{attribute 'linkalways'} 
{attribute 'no_explicit_call' := 'This FB is a CLASS and must be accessed using methods or properties'}
{attribute 'enable_dynamic_creation'}
FUNCTION_BLOCK Node_F_VN_EnclosingTriangle EXTENDS VisionNode
VAR
    ipPointSet : _ITcVnContainer;
    aTriangleVertices : _TcVnArray3_Point2_REAL;
    fArea : _LREAL(0.0);
    hrPrev : _HRESULT(S_OK);
	hresult : _HRESULT(S_OK);
END_VAR

METHOD PUBLIC  Clone : I_Node
VAR
	pNode : POINTER TO Node_F_VN_EnclosingTriangle;
END_VAR
pNode := __NEW(Node_F_VN_EnclosingTriangle);
Clone := pNode^;
END_METHOD

METHOD FB_init : BOOL
VAR_INPUT
	bInitRetains : BOOL; // if TRUE, the retain variables are initialized (warm start / cold start)
	bInCopyCode : BOOL;  // if TRUE, the instance afterwards gets moved into the copy code (online change)
END_VAR
AddInput('ipPointSet', ipPointSet);
AddInput('hrPrev', hrPrev);
AddOutput('aTriangleVertices', aTriangleVertices);
AddOutput('fArea', fArea);
AddOutput('hresult',hresult);
END_METHOD

METHOD PROTECTED OnExecute
VAR
    area : LREAL;
END_VAR
hresult.Value := F_VN_EnclosingTriangle(
	ipPointSet := ipPointSet.Value,
    aTriangleVertices := aTriangleVertices.Value,
	hrPrev:= hrPrev.Value,
    fArea => area);

IF SUCCEEDED(hresult.Value) THEN
    fArea.Value := area;
END_IF
END_METHOD

METHOD PUBLIC PreExecutionCheck
VAR_INPUT
	Check : I_PreExecutionChecks;
END_VAR
Check.IsTrue(ipPointSet.IsValid, 'ipPointSet must be a valid container');
Check.IsTrue((ipPointSet.IsType(TC_GLOBAL_CONST_LIST.ContainerType_Vector_TcVnPoint2_DINT) OR
              ipPointSet.IsType(TC_GLOBAL_CONST_LIST.ContainerType_Vector_TcVnPoint2_REAL)),
              'ipPointSet contains incorrect type');
END_METHOD

END_FUNCTION_BLOCK

(* stored: Version 1.1.0.1, ProductVersion 3.1.4026.13
   POU Node_F_VN_EnclosingTriangle: Id {111ed582-313e-0d05-2789-6f60a7664767}, SpecialFunc None
   Folder Constructor: Id {3620c78e-60ad-0497-028c-3a083e9bf22e}
   Method Clone: Id {33645f09-07c7-0d26-2a84-af710fbc05a7}
   Method FB_init: Id {525f8962-5e73-069c-08e4-c1e55d76f4cd}
   Method OnExecute: Id {a579b5e4-6b47-00ea-3de1-cde018662825}
   Method PreExecutionCheck: Id {310e661c-25fe-062c-3ceb-325b67e876ef} *)
